(* Logix 5000 project; controller Amvex_Thorpe_Flowmeter vendor 1 type 14 code 106 rev 33.13; software revision 33.01; part 3 of 16 *)

ADD_ON_INSTRUCTION MoveJoints   (* revision 0.1, vendor Mecademic Inc., ExecuteEnableInFalse *)
// Move each joint to given absolute position in degrees
VAR_IN_OUT
   RobotInputs : _061D:Meca500_86BDA20B:I:0; {required}
   RobotOutputs : _061D:Meca500_01F88326:O:0; {required}
END_VAR
VAR_INPUT
   Joint_1_Angle : REAL; {required}
   Joint_2_Angle : REAL; {required}
   Joint_3_Angle : REAL; {required}
   Joint_4_Angle : REAL; {required}
   Joint_5_Angle : REAL; {required}
   Joint_6_Angle : REAL; {required}
   ExternalStateControl : BOOL; {required}
   ExternalMoveID : INT; {required}
END_VAR
VAR_OUTPUT
   Enabled : BOOL; {visible}
   Sent : BOOL; {visible}
   Buffered : BOOL; {visible}
   Error : BOOL; {visible}
END_VAR
VAR
   InternalMoveID : INT; {access None}
   MoveIDUpdated : BOOL; {access None}
   OneShot : DINT; {access None}
   MoveIDTrig : BOOL; {access None}
   FirstScan : BOOL; {access None}
END_VAR

ROUTINE EnableInFalse   (* ladder *)
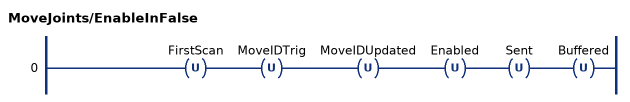
   0: OTU(FirstScan)OTU(MoveIDTrig)OTU(MoveIDUpdated)OTU(Enabled)OTU(Sent)OTU(Buffered);
END_ROUTINE

ROUTINE Logic   (* ladder *)
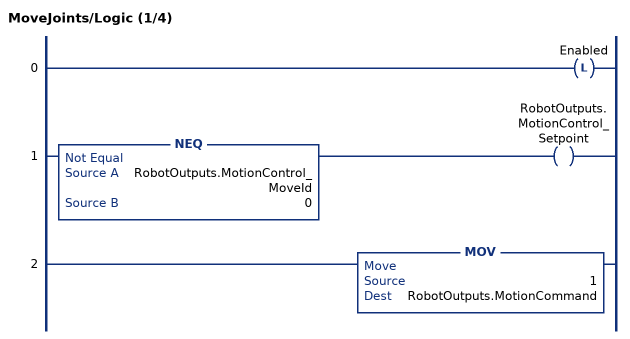
   0: OTL(Enabled);
   1: NEQ(RobotOutputs.MotionControl_MoveId,0)OTE(RobotOutputs.MotionControl_Setpoint);
   2: MOV(1,RobotOutputs.MotionCommand);
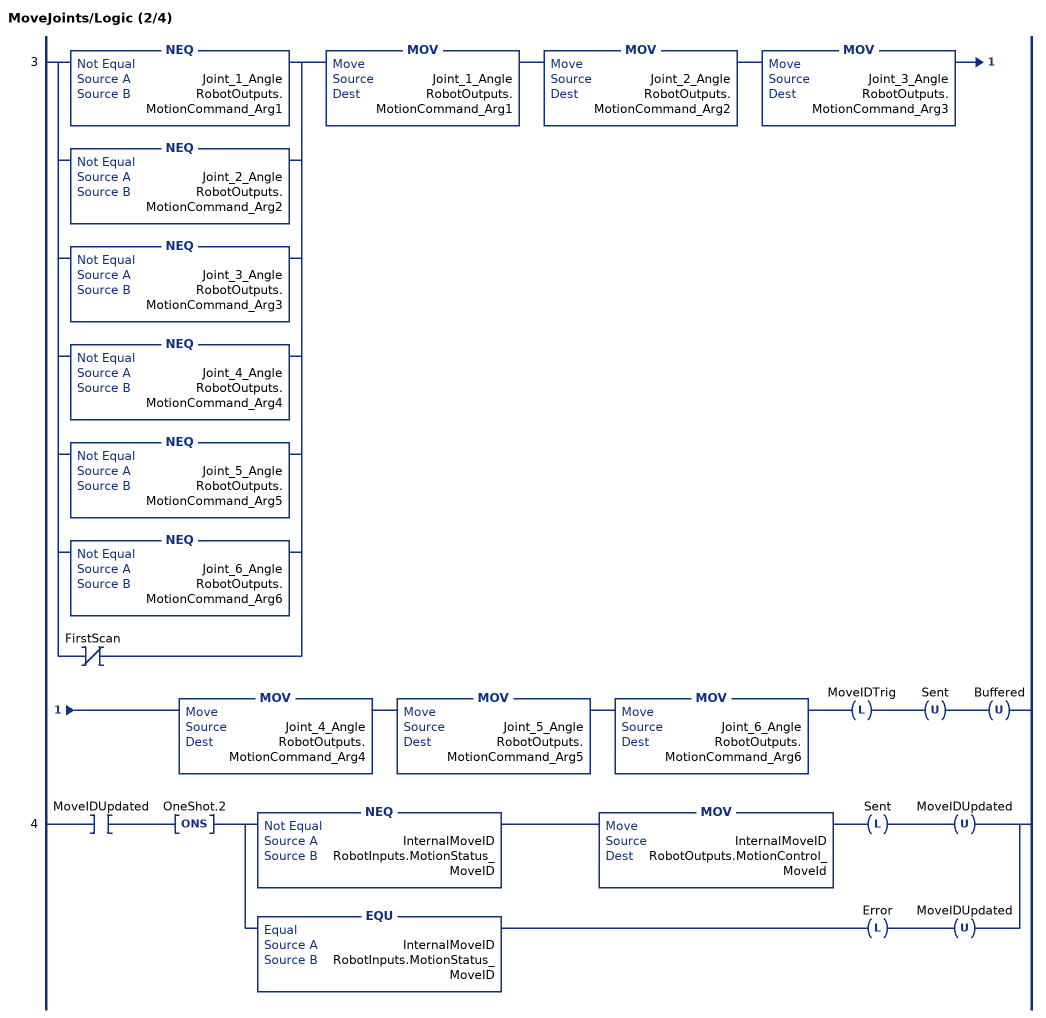
   3: [NEQ(Joint_1_Angle,RobotOutputs.MotionCommand_Arg1) ,NEQ(Joint_2_Angle,RobotOutputs.MotionCommand_Arg2) ,NEQ(Joint_3_Angle,RobotOutputs.MotionCommand_Arg3) ,NEQ(Joint_4_Angle,RobotOutputs.MotionCommand_Arg4) ,NEQ(Joint_5_Angle,RobotOutputs.MotionCommand_Arg5) ,NEQ(Joint_6_Angle,RobotOutputs.MotionCommand_Arg6) ,XIO(FirstScan) ]MOV(Joint_1_Angle,RobotOutputs.MotionCommand_Arg1)MOV(Joint_2_Angle,RobotOutputs.MotionCommand_Arg2)MOV(Joint_3_Angle,RobotOutputs.MotionCommand_Arg3)MOV(Joint_4_Angle,RobotOutputs.MotionCommand_Arg4)MOV(Joint_5_Angle,RobotOutputs.MotionCommand_Arg5)MOV(Joint_6_Angle,RobotOutputs.MotionCommand_Arg6)OTL(MoveIDTrig)OTU(Sent)OTU(Buffered);
   4: XIC(MoveIDUpdated)ONS(OneShot.2)[NEQ(InternalMoveID,RobotInputs.MotionStatus_MoveID) MOV(InternalMoveID,RobotOutputs.MotionControl_MoveId) OTL(Sent) OTU(MoveIDUpdated) ,EQU(InternalMoveID,RobotInputs.MotionStatus_MoveID) OTL(Error) OTU(MoveIDUpdated) ];
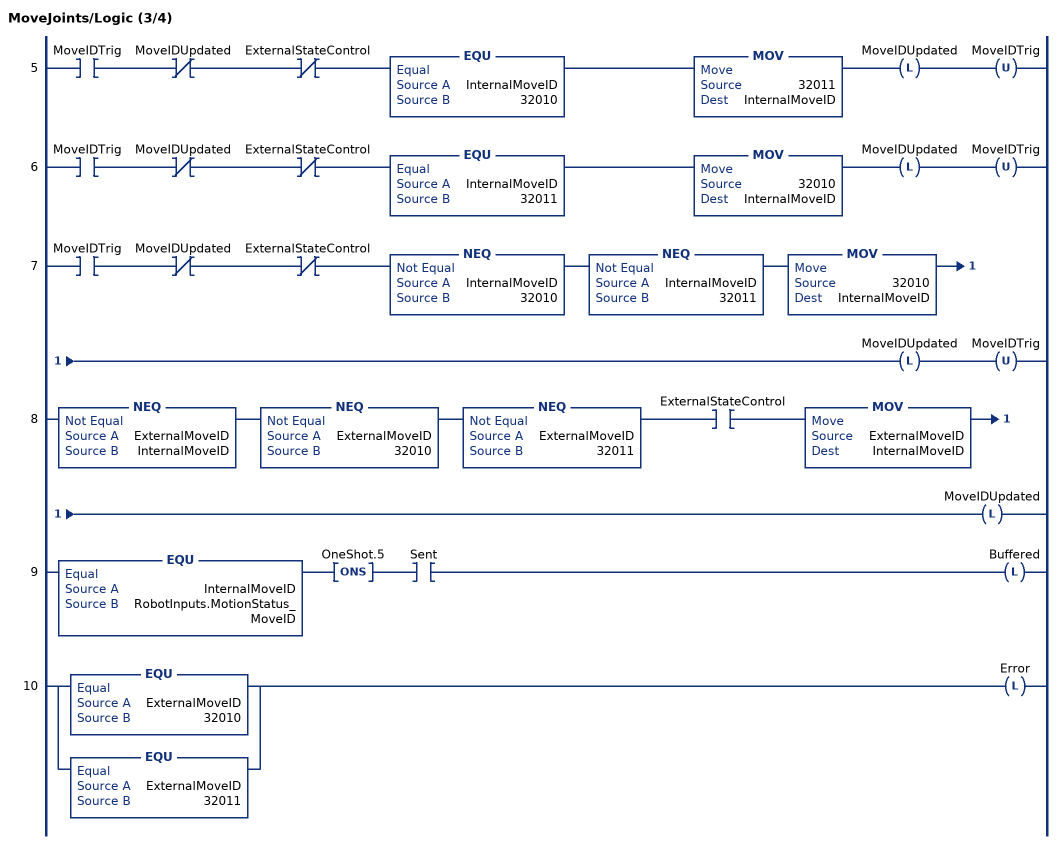
   5: XIC(MoveIDTrig)XIO(MoveIDUpdated)XIO(ExternalStateControl)EQU(InternalMoveID,32010)MOV(32011,InternalMoveID)OTL(MoveIDUpdated)OTU(MoveIDTrig);
   6: XIC(MoveIDTrig)XIO(MoveIDUpdated)XIO(ExternalStateControl)EQU(InternalMoveID,32011)MOV(32010,InternalMoveID)OTL(MoveIDUpdated)OTU(MoveIDTrig);
   7: XIC(MoveIDTrig)XIO(MoveIDUpdated)XIO(ExternalStateControl)NEQ(InternalMoveID,32010)NEQ(InternalMoveID,32011)MOV(32010,InternalMoveID)OTL(MoveIDUpdated)OTU(MoveIDTrig);
   8: NEQ(ExternalMoveID,InternalMoveID)NEQ(ExternalMoveID,32010)NEQ(ExternalMoveID,32011)XIC(ExternalStateControl)MOV(ExternalMoveID,InternalMoveID)OTL(MoveIDUpdated);
   9: EQU(InternalMoveID,RobotInputs.MotionStatus_MoveID)ONS(OneShot.5)XIC(Sent)OTL(Buffered);
   10: [EQU(ExternalMoveID,32010) ,EQU(ExternalMoveID,32011) ]OTL(Error);
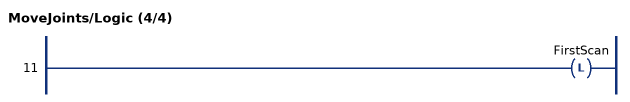
   11: OTL(FirstScan);
END_ROUTINE
END_ADD_ON_INSTRUCTION

ADD_ON_INSTRUCTION MoveJointsRel   (* revision 1.0, vendor Mecademic inc., ExecuteEnableInFalse *)
// Move each joint relative to current robot position
VAR_IN_OUT
   RobotOutputs : _061D:Meca500_01F88326:O:0; {required}
   RobotInputs : _061D:Meca500_86BDA20B:I:0; {required}
END_VAR
VAR_INPUT
   Angle_Joint_1 : REAL; {required}   // [-350..350]
   Angle_Joint_2 : REAL; {required}   // [-160..160}
   Angle_Joint_3 : REAL; {required}   // [-205..205]
   Angle_Joint_4 : REAL; {required}   // [-340..340]
   Angle_Joint_5 : REAL; {required}   // [-230..230]
   Angle_Joint_6 : REAL; {required}   // [-72000..72000]
   ExternalStateControl : BOOL; {required}
   ExternalMoveID : INT; {required}
END_VAR
VAR_OUTPUT
   Enabled : BOOL; {access Read Only, visible}
   Sent : BOOL; {access Read Only, visible}
   Error : BOOL; {access Read Only, visible}
   Buffered : BOOL; {access Read Only, visible}
END_VAR
VAR
   FirstScan : BOOL; {access None}
   MoveIDUpdated : BOOL; {access None}
   OneShot : DINT; {access None}
   InternalMoveID : DINT; {access None}
   MoveIDTrig : BOOL; {access None}
END_VAR

ROUTINE EnableInFalse   (* ladder *)
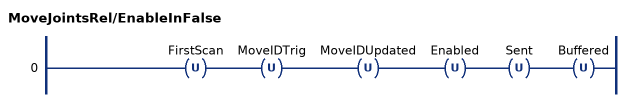
   0: OTU(FirstScan)OTU(MoveIDTrig)OTU(MoveIDUpdated)OTU(Enabled)OTU(Sent)OTU(Buffered);
END_ROUTINE

ROUTINE Logic   (* ladder *)
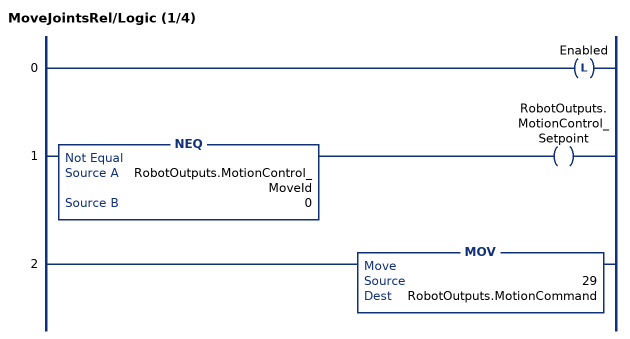
   0: OTL(Enabled);
   1: NEQ(RobotOutputs.MotionControl_MoveId,0)OTE(RobotOutputs.MotionControl_Setpoint);
   2: MOV(29,RobotOutputs.MotionCommand);
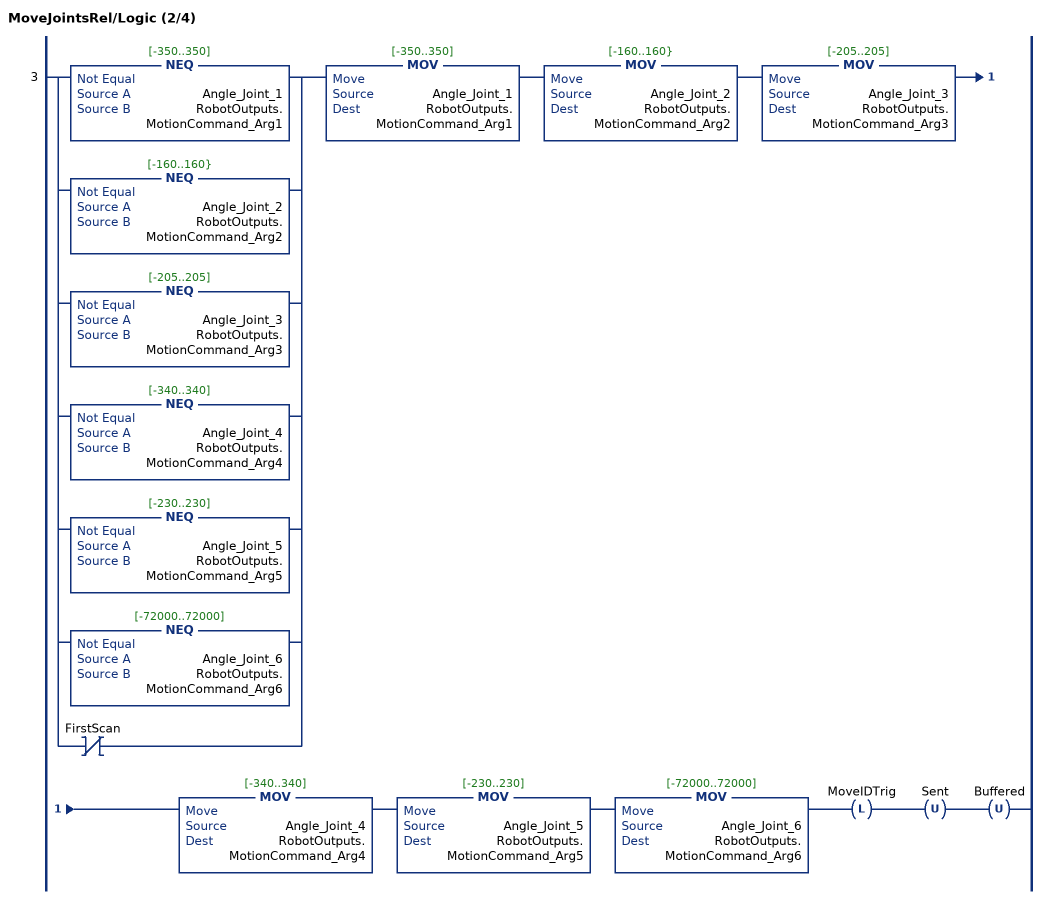
   3: [NEQ(Angle_Joint_1,RobotOutputs.MotionCommand_Arg1) ,NEQ(Angle_Joint_2,RobotOutputs.MotionCommand_Arg2) ,NEQ(Angle_Joint_3,RobotOutputs.MotionCommand_Arg3) ,NEQ(Angle_Joint_4,RobotOutputs.MotionCommand_Arg4) ,NEQ(Angle_Joint_5,RobotOutputs.MotionCommand_Arg5) ,NEQ(Angle_Joint_6,RobotOutputs.MotionCommand_Arg6) ,XIO(FirstScan) ]MOV(Angle_Joint_1,RobotOutputs.MotionCommand_Arg1)MOV(Angle_Joint_2,RobotOutputs.MotionCommand_Arg2)MOV(Angle_Joint_3,RobotOutputs.MotionCommand_Arg3)MOV(Angle_Joint_4,RobotOutputs.MotionCommand_Arg4)MOV(Angle_Joint_5,RobotOutputs.MotionCommand_Arg5)MOV(Angle_Joint_6,RobotOutputs.MotionCommand_Arg6)OTL(MoveIDTrig)OTU(Sent)OTU(Buffered);
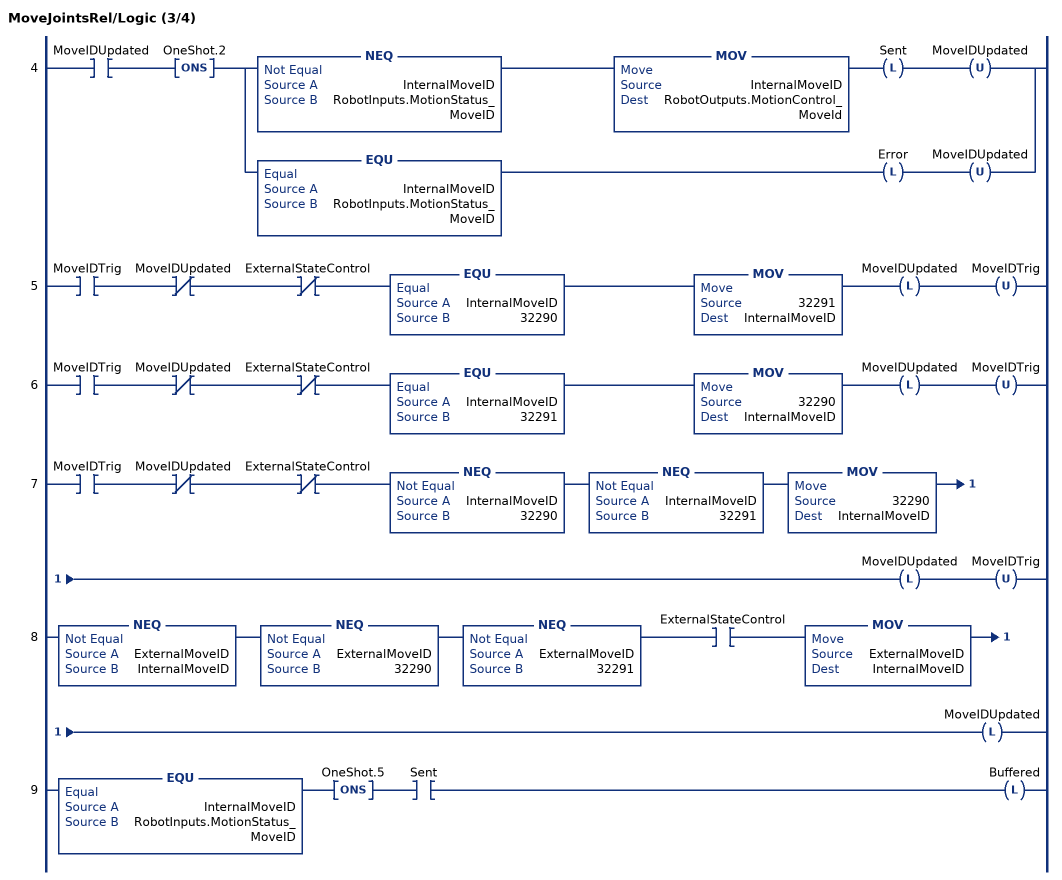
   4: XIC(MoveIDUpdated)ONS(OneShot.2)[NEQ(InternalMoveID,RobotInputs.MotionStatus_MoveID) MOV(InternalMoveID,RobotOutputs.MotionControl_MoveId) OTL(Sent) OTU(MoveIDUpdated) ,EQU(InternalMoveID,RobotInputs.MotionStatus_MoveID) OTL(Error) OTU(MoveIDUpdated) ];
   5: XIC(MoveIDTrig)XIO(MoveIDUpdated)XIO(ExternalStateControl)EQU(InternalMoveID,32290)MOV(32291,InternalMoveID)OTL(MoveIDUpdated)OTU(MoveIDTrig);
   6: XIC(MoveIDTrig)XIO(MoveIDUpdated)XIO(ExternalStateControl)EQU(InternalMoveID,32291)MOV(32290,InternalMoveID)OTL(MoveIDUpdated)OTU(MoveIDTrig);
   7: XIC(MoveIDTrig)XIO(MoveIDUpdated)XIO(ExternalStateControl)NEQ(InternalMoveID,32290)NEQ(InternalMoveID,32291)MOV(32290,InternalMoveID)OTL(MoveIDUpdated)OTU(MoveIDTrig);
   8: NEQ(ExternalMoveID,InternalMoveID)NEQ(ExternalMoveID,32290)NEQ(ExternalMoveID,32291)XIC(ExternalStateControl)MOV(ExternalMoveID,InternalMoveID)OTL(MoveIDUpdated);
   9: EQU(InternalMoveID,RobotInputs.MotionStatus_MoveID)ONS(OneShot.5)XIC(Sent)OTL(Buffered);
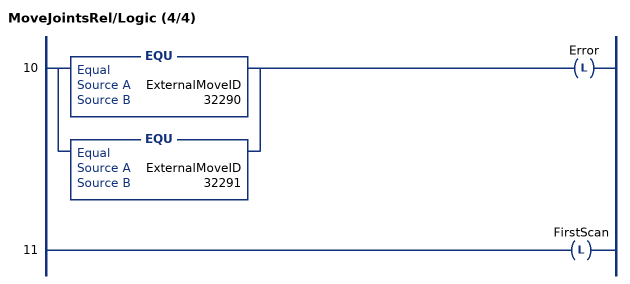
   10: [EQU(ExternalMoveID,32290) ,EQU(ExternalMoveID,32291) ]OTL(Error);
   11: OTL(FirstScan);
END_ROUTINE
END_ADD_ON_INSTRUCTION

ADD_ON_INSTRUCTION MoveJointsVel   (* revision 0.1, vendor Mecademic Inc., ExecuteEnableInFalse *)
// Set current mode to "join velocity mode"
VAR_IN_OUT
   RobotInputs : _061D:Meca500_86BDA20B:I:0; {required}
   RobotOutputs : _061D:Meca500_01F88326:O:0; {required}
END_VAR
VAR_INPUT
   Joint_1_Vel : REAL; {required}
   Joint_2_Vel : REAL; {required}
   Joint_3_Vel : REAL; {required}
   Joint_4_Vel : REAL; {required}
   Joint_5_Vel : REAL; {required}
   Joint_6_Vel : REAL; {required}
   ExternalStateControl : BOOL; {required}
   ExternalMoveID : INT; {required}
END_VAR
VAR_OUTPUT
   Enabled : BOOL; {visible}
   Sent : BOOL; {visible}
   Buffered : BOOL; {visible}
   Error : BOOL; {visible}
END_VAR
VAR
   InternalMoveID : INT; {access None}
   MoveIDTrig : BOOL; {access None}
   MoveIDUpdated : BOOL; {access None}
   OneShot : DINT; {access None}
   FirstScan : BOOL; {access None}
END_VAR

ROUTINE EnableInFalse   (* ladder *)
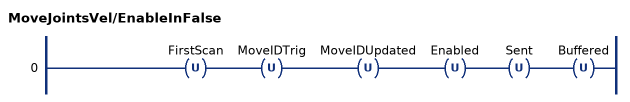
   0: OTU(FirstScan)OTU(MoveIDTrig)OTU(MoveIDUpdated)OTU(Enabled)OTU(Sent)OTU(Buffered);
END_ROUTINE

ROUTINE Logic   (* ladder *)
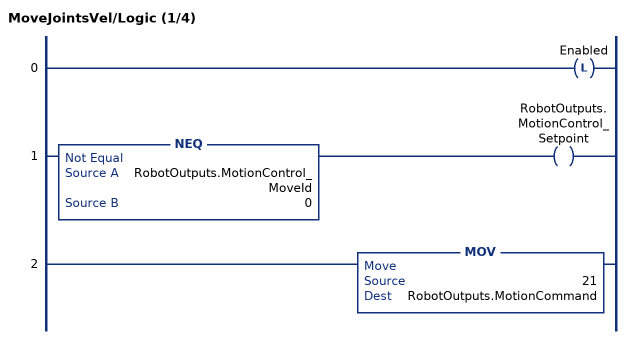
   0: OTL(Enabled);
   1: NEQ(RobotOutputs.MotionControl_MoveId,0)OTE(RobotOutputs.MotionControl_Setpoint);
   2: MOV(21,RobotOutputs.MotionCommand);
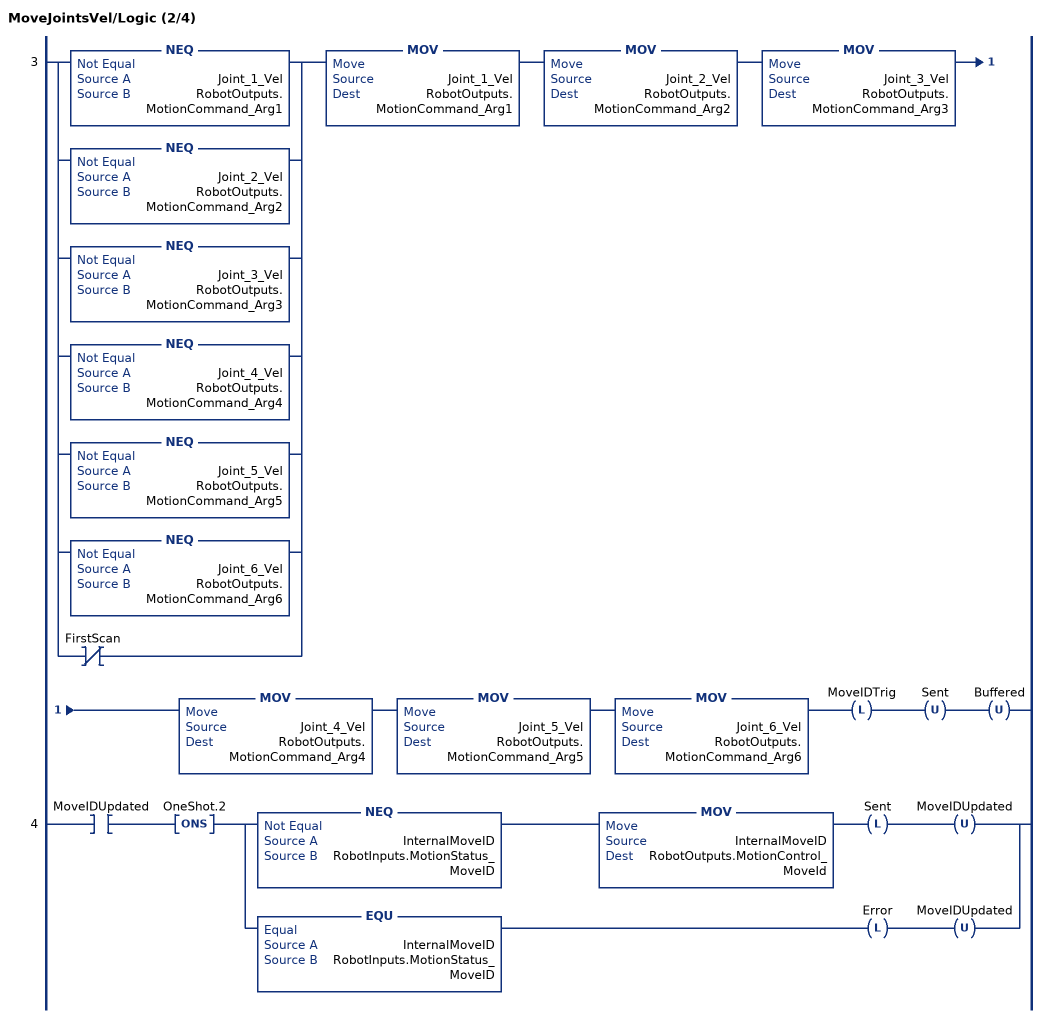
   3: [NEQ(Joint_1_Vel,RobotOutputs.MotionCommand_Arg1) ,NEQ(Joint_2_Vel,RobotOutputs.MotionCommand_Arg2) ,NEQ(Joint_3_Vel,RobotOutputs.MotionCommand_Arg3) ,NEQ(Joint_4_Vel,RobotOutputs.MotionCommand_Arg4) ,NEQ(Joint_5_Vel,RobotOutputs.MotionCommand_Arg5) ,NEQ(Joint_6_Vel,RobotOutputs.MotionCommand_Arg6) ,XIO(FirstScan) ]MOV(Joint_1_Vel,RobotOutputs.MotionCommand_Arg1)MOV(Joint_2_Vel,RobotOutputs.MotionCommand_Arg2)MOV(Joint_3_Vel,RobotOutputs.MotionCommand_Arg3)MOV(Joint_4_Vel,RobotOutputs.MotionCommand_Arg4)MOV(Joint_5_Vel,RobotOutputs.MotionCommand_Arg5)MOV(Joint_6_Vel,RobotOutputs.MotionCommand_Arg6)OTL(MoveIDTrig)OTU(Sent)OTU(Buffered);
   4: XIC(MoveIDUpdated)ONS(OneShot.2)[NEQ(InternalMoveID,RobotInputs.MotionStatus_MoveID) MOV(InternalMoveID,RobotOutputs.MotionControl_MoveId) OTL(Sent) OTU(MoveIDUpdated) ,EQU(InternalMoveID,RobotInputs.MotionStatus_MoveID) OTL(Error) OTU(MoveIDUpdated) ];
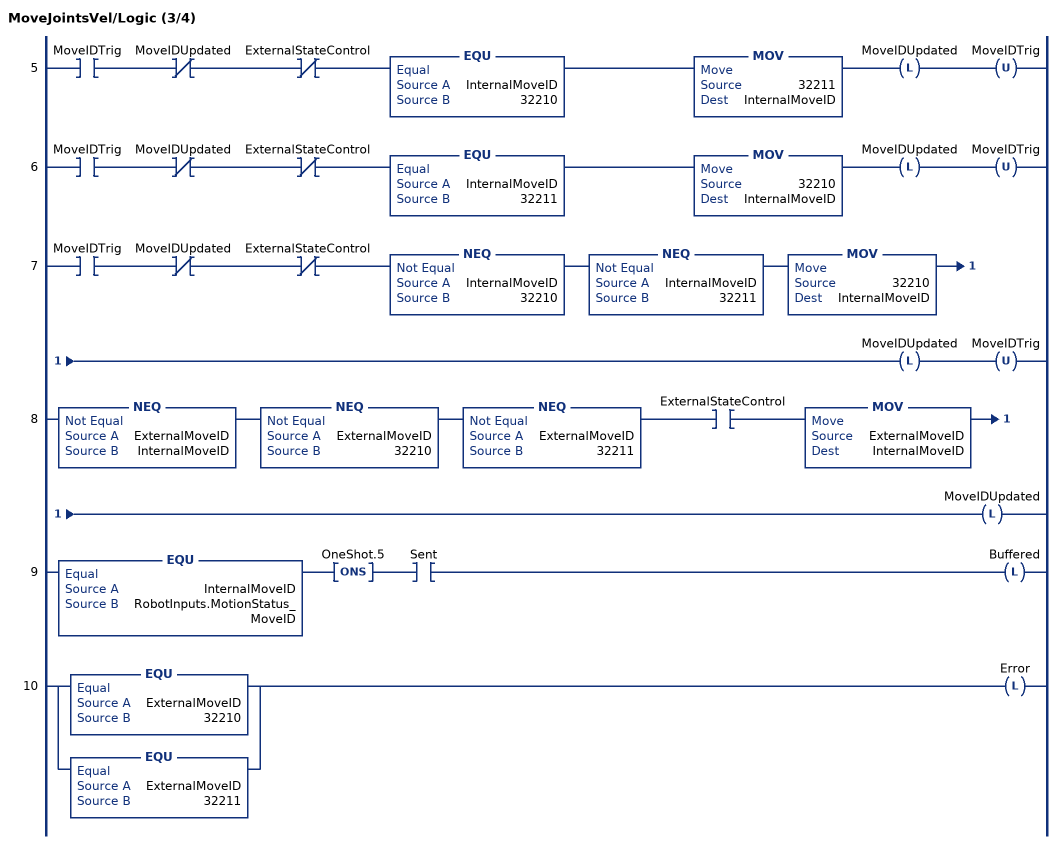
   5: XIC(MoveIDTrig)XIO(MoveIDUpdated)XIO(ExternalStateControl)EQU(InternalMoveID,32210)MOV(32211,InternalMoveID)OTL(MoveIDUpdated)OTU(MoveIDTrig);
   6: XIC(MoveIDTrig)XIO(MoveIDUpdated)XIO(ExternalStateControl)EQU(InternalMoveID,32211)MOV(32210,InternalMoveID)OTL(MoveIDUpdated)OTU(MoveIDTrig);
   7: XIC(MoveIDTrig)XIO(MoveIDUpdated)XIO(ExternalStateControl)NEQ(InternalMoveID,32210)NEQ(InternalMoveID,32211)MOV(32210,InternalMoveID)OTL(MoveIDUpdated)OTU(MoveIDTrig);
   8: NEQ(ExternalMoveID,InternalMoveID)NEQ(ExternalMoveID,32210)NEQ(ExternalMoveID,32211)XIC(ExternalStateControl)MOV(ExternalMoveID,InternalMoveID)OTL(MoveIDUpdated);
   9: EQU(InternalMoveID,RobotInputs.MotionStatus_MoveID)ONS(OneShot.5)XIC(Sent)OTL(Buffered);
   10: [EQU(ExternalMoveID,32210) ,EQU(ExternalMoveID,32211) ]OTL(Error);
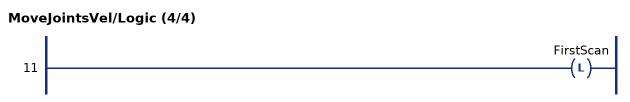
   11: OTL(FirstScan);
END_ROUTINE
END_ADD_ON_INSTRUCTION

ADD_ON_INSTRUCTION MoveLin   (* revision 0.1, vendor Mecademic Inc., ExecuteEnableInFalse *)
// Move to a position relative to WRF (x-y-z in mm, a-b-c in degrees). Movement of the tool is linear in space (follows a straight line)
VAR_IN_OUT
   RobotInputs : _061D:Meca500_86BDA20B:I:0; {required}
   RobotOutputs : _061D:Meca500_01F88326:O:0; {required}
END_VAR
VAR_INPUT
   Pose_X_Pos : REAL; {required}
   Pose_Y_Pos : REAL; {required}
   Pose_Z_Pos : REAL; {required}
   Pose_rX_Ang : REAL; {required}
   Pose_rY_Ang : REAL; {required}
   Pose_rZ_Ang : REAL; {required}
   ExternalStateControl : BOOL; {required}
   ExternalMoveID : INT; {required}
END_VAR
VAR_OUTPUT
   Enabled : BOOL; {visible}
   Sent : BOOL; {visible}
   Buffered : BOOL; {visible}
   Error : BOOL; {visible}
END_VAR
VAR
   InternalMoveID : INT; {access None}
   MoveIDTrig : BOOL; {access None}
   MoveIDUpdated : BOOL; {access None}
   OneShot : DINT; {access None}
   FirstScan : BOOL; {access None}
END_VAR

ROUTINE EnableInFalse   (* ladder *)
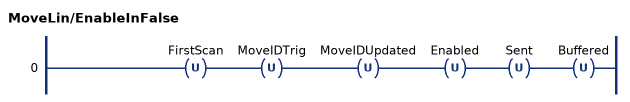
   0: OTU(FirstScan)OTU(MoveIDTrig)OTU(MoveIDUpdated)OTU(Enabled)OTU(Sent)OTU(Buffered);
END_ROUTINE

ROUTINE Logic   (* ladder *)
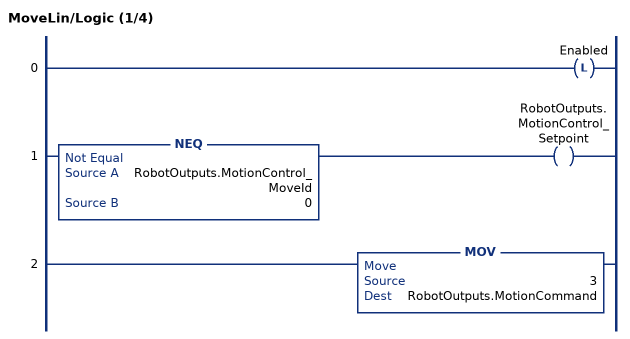
   0: OTL(Enabled);
   1: NEQ(RobotOutputs.MotionControl_MoveId,0)OTE(RobotOutputs.MotionControl_Setpoint);
   2: MOV(3,RobotOutputs.MotionCommand);
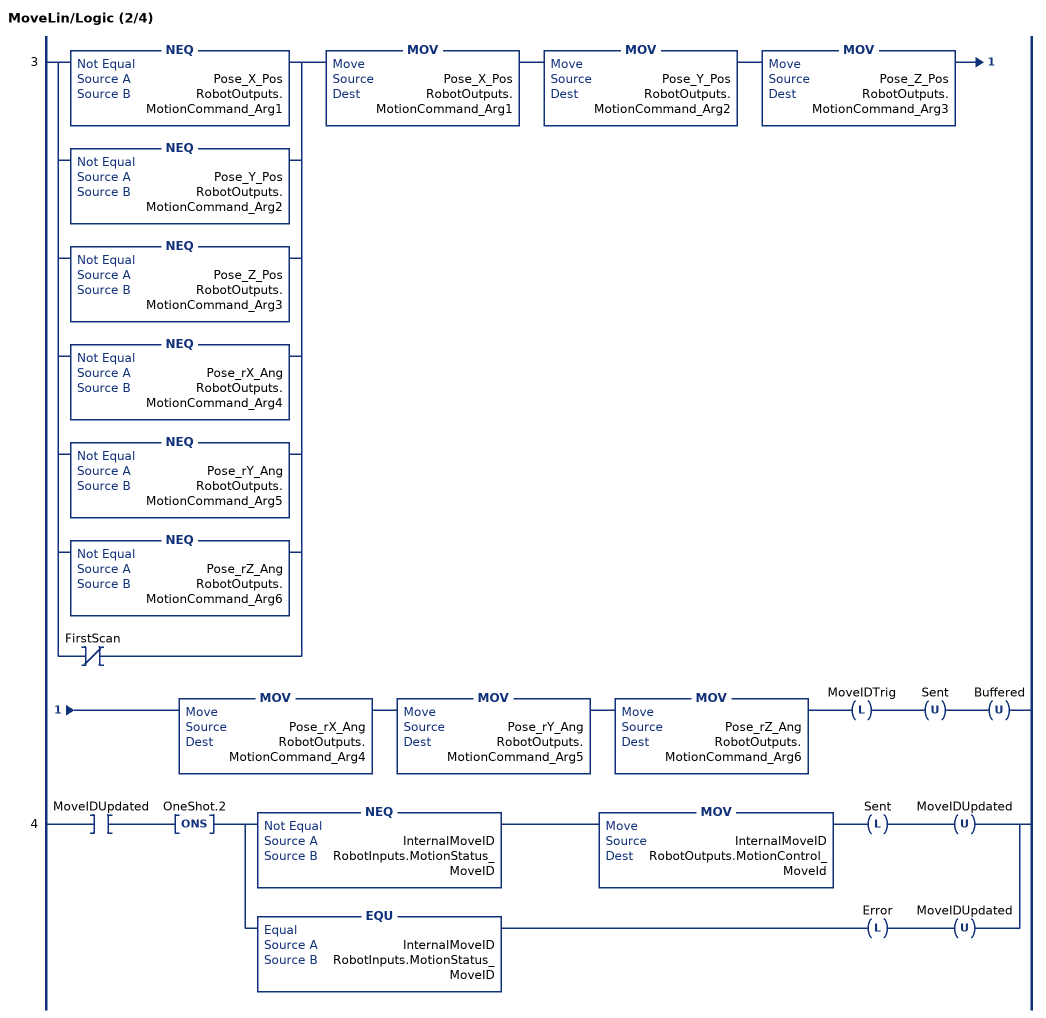
   3: [NEQ(Pose_X_Pos,RobotOutputs.MotionCommand_Arg1) ,NEQ(Pose_Y_Pos,RobotOutputs.MotionCommand_Arg2) ,NEQ(Pose_Z_Pos,RobotOutputs.MotionCommand_Arg3) ,NEQ(Pose_rX_Ang,RobotOutputs.MotionCommand_Arg4) ,NEQ(Pose_rY_Ang,RobotOutputs.MotionCommand_Arg5) ,NEQ(Pose_rZ_Ang,RobotOutputs.MotionCommand_Arg6) ,XIO(FirstScan) ]MOV(Pose_X_Pos,RobotOutputs.MotionCommand_Arg1)MOV(Pose_Y_Pos,RobotOutputs.MotionCommand_Arg2)MOV(Pose_Z_Pos,RobotOutputs.MotionCommand_Arg3)MOV(Pose_rX_Ang,RobotOutputs.MotionCommand_Arg4)MOV(Pose_rY_Ang,RobotOutputs.MotionCommand_Arg5)MOV(Pose_rZ_Ang,RobotOutputs.MotionCommand_Arg6)OTL(MoveIDTrig)OTU(Sent)OTU(Buffered);
   4: XIC(MoveIDUpdated)ONS(OneShot.2)[NEQ(InternalMoveID,RobotInputs.MotionStatus_MoveID) MOV(InternalMoveID,RobotOutputs.MotionControl_MoveId) OTL(Sent) OTU(MoveIDUpdated) ,EQU(InternalMoveID,RobotInputs.MotionStatus_MoveID) OTL(Error) OTU(MoveIDUpdated) ];
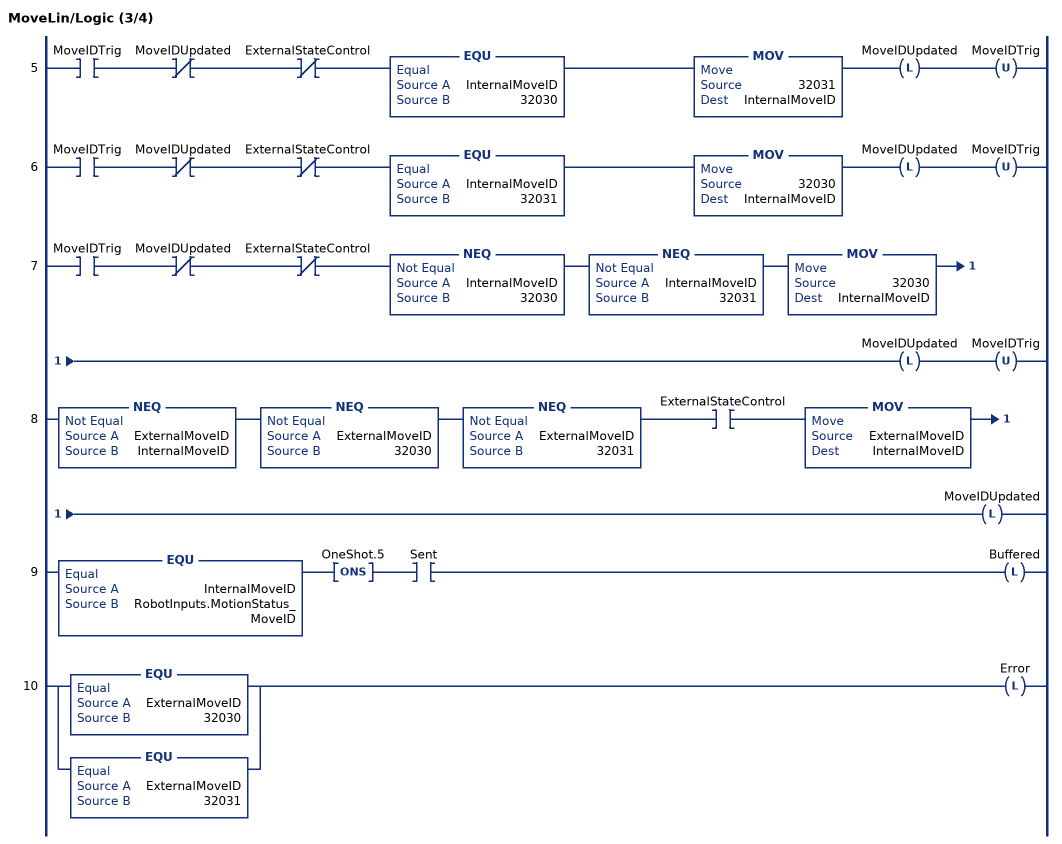
   5: XIC(MoveIDTrig)XIO(MoveIDUpdated)XIO(ExternalStateControl)EQU(InternalMoveID,32030)MOV(32031,InternalMoveID)OTL(MoveIDUpdated)OTU(MoveIDTrig);
   6: XIC(MoveIDTrig)XIO(MoveIDUpdated)XIO(ExternalStateControl)EQU(InternalMoveID,32031)MOV(32030,InternalMoveID)OTL(MoveIDUpdated)OTU(MoveIDTrig);
   7: XIC(MoveIDTrig)XIO(MoveIDUpdated)XIO(ExternalStateControl)NEQ(InternalMoveID,32030)NEQ(InternalMoveID,32031)MOV(32030,InternalMoveID)OTL(MoveIDUpdated)OTU(MoveIDTrig);
   8: NEQ(ExternalMoveID,InternalMoveID)NEQ(ExternalMoveID,32030)NEQ(ExternalMoveID,32031)XIC(ExternalStateControl)MOV(ExternalMoveID,InternalMoveID)OTL(MoveIDUpdated);
   9: EQU(InternalMoveID,RobotInputs.MotionStatus_MoveID)ONS(OneShot.5)XIC(Sent)OTL(Buffered);
   10: [EQU(ExternalMoveID,32030) ,EQU(ExternalMoveID,32031) ]OTL(Error);
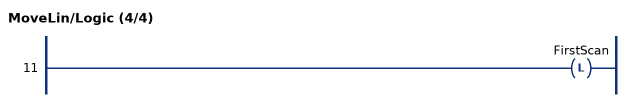
   11: OTL(FirstScan);
END_ROUTINE
END_ADD_ON_INSTRUCTION
